// TwinCAT 3 PLC project liftConv
// ProgramVersion: 3.1.0.9
// libraries:
//   VisuElem3DPath, 3.5.6.0 (System)
//   VisuElemMeter, 3.5.6.0 (System)
//   VisuElems, 3.5.6.10 (System)
//   VisuElemsDateTime, 3.5.6.0 (System)
//   VisuElemsSpecialControls, 3.5.6.0 (System)
//   VisuElemsWinControls, 3.5.6.0 (System)
//   VisuElemTextEditor, 3.5.6.0 (System)
//   visuinputs, 3.5.6.0 (system)
//   VisuNativeControl, 3.5.6.0 (System)
//   Tc2_Standard, * (Beckhoff Automation GmbH)
//   Tc2_System, * (Beckhoff Automation GmbH)
//   Tc3_Interfaces, * (Beckhoff Automation GmbH)
//   Tc3_Module, * (Beckhoff Automation GmbH)
//   VisuDialogs, * (System)
// project tree:
//   / GlobalTextList.TcGTLO, PlcTask.TcTTO, Visualization Manager.TcVMO (not stored), VISU_TASK.TcTTO
//   GVLs/ GVL.TcGVL
//   POUs/ MAIN.TcPOU, outputFBD.TcPOU, NotUsed.TcPOU, Queues.TcPOU, resetOutputs.TcPOU, reset.TcPOU
//   VISUs/ TouchScreen.TcVIS
// real-time tasks:
//   TASK PlcTask: cycle T#10ms, priority 20, ADS port 350
//   TASK VISU_TASK: cycle T#100000us, priority 30, ADS port 351
// I/O:
//   DEVICE Device 1 (EtherCAT), AmsNetId 5.29.55.232.2.1
//     Term 1 (EK1100) [EK1100 EtherCAT Coupler (2A E-Bus)]
//       Term 2 (EL1008) [EL1008 8Ch. Dig. Input 24V, 3ms]
//       Term 3 (EL2008) [EL2008 8Ch. Dig. Output 24V, 0.5A]
//       Term 4 (EL3002) [EL3002 2Ch. Ana. Input +/-10V]
//       Term 5 (EL4002) [EL4002 2Ch. Ana. Output 0-10V, 12bit]
//       Term 6 (EL3124) [EL3124 4Ch. Ana. Input 4-20mA Diff.]
//       Term 7 (EL4024) [EL4024 4Ch. Ana. Output 4-20mA, 12bit]
//       Term 10 (EL9011) [EL9011 End Terminal]
//     Term 8 (EK1100) [EK1100 EtherCAT Coupler (2A E-Bus)]
//       Box 9 (BK1250)
// variable links:
//   liftConv/liftConv Instance <-> Device 1 (EtherCAT)/Term 1 (EK1100)/Term 2 (EL1008)
//     PlcTask Inputs/GVL.b{1..5} <-> Channel {1..5}/Input  (5 links)
//   liftConv/liftConv Instance <-> Device 1 (EtherCAT)/Term 8 (EK1100)/Box 9 (BK1250)
//     PlcTask Inputs/GVL.I_bInput11 <-> Term 4 (KL1104)/Channel 3/Input
//     PlcTask Inputs/GVL.I_bInput12 <-> Term 4 (KL1104)/Channel 4/Input
//     PlcTask Inputs/GVL.bottomLeft_IB <-> Term 4 (KL1104)/Channel 1/Input
//     PlcTask Inputs/GVL.bottomRight_IB <-> Term 3 (KL1104)/Channel 3/Input
//     PlcTask Inputs/GVL.leftLiftDownPosition_IB <-> Term 3 (KL1104)/Channel 2/Input
//     PlcTask Inputs/GVL.leftLiftOptical_IB <-> Term 2 (KL1104)/Channel 1/Input
//     PlcTask Inputs/GVL.leftLiftUpPosition_IB <-> Term 3 (KL1104)/Channel 1/Input
//     PlcTask Inputs/GVL.rightLiftDownPosition_IB <-> Term 2 (KL1104)/Channel 4/Input
//     PlcTask Inputs/GVL.rightLiftOptical_IB <-> Term 2 (KL1104)/Channel 2/Input
//     PlcTask Inputs/GVL.rightLiftUpPosition_IB <-> Term 2 (KL1104)/Channel 3/Input
//     PlcTask Inputs/GVL.topLeft_IB <-> Term 4 (KL1104)/Channel 2/Input
//     PlcTask Inputs/GVL.topRight_IB <-> Term 3 (KL1104)/Channel 4/Input
//     PlcTask Outputs/GVL.bottomBeltRight_OB <-> Term 7 (KL2114)/Channel 2/Output
//     PlcTask Outputs/GVL.leftLiftBeltLeft_OB <-> Term 6 (KL2114)/Channel 4/Output
//     PlcTask Outputs/GVL.leftLiftBeltRight_OB <-> Term 6 (KL2114)/Channel 3/Output
//     PlcTask Outputs/GVL.leftLiftDown_OB <-> Term 5 (KL2114)/Channel 2/Output
//     PlcTask Outputs/GVL.leftLiftUp_OB <-> Term 5 (KL2114)/Channel 1/Output
//     PlcTask Outputs/GVL.rightLiftBeltLeft_OB <-> Term 6 (KL2114)/Channel 1/Output
//     PlcTask Outputs/GVL.rightLiftBeltRight_OB <-> Term 6 (KL2114)/Channel 2/Output
//     PlcTask Outputs/GVL.rightLiftDown_OB <-> Term 5 (KL2114)/Channel 3/Output
//     PlcTask Outputs/GVL.rightLiftUp_OB <-> Term 5 (KL2114)/Channel 4/Output
//     PlcTask Outputs/GVL.topBeltLeft_OB <-> Term 7 (KL2114)/Channel 1/Output

CONFIGURATION liftConv
    RESOURCE PLC ON TwinCAT3
        TASK PlcTask(INTERVAL := T#10ms, PRIORITY := 20);
        TASK VISU_TASK(INTERVAL := T#100000us, PRIORITY := 30);
        PROGRAM MAIN WITH PlcTask : MAIN;
        PROGRAM VisuElems_Visu_Prg WITH VISU_TASK : VisuElems.Visu_Prg;
    END_RESOURCE
END_CONFIGURATION

// ---- GVLs/GVL.TcGVL
VAR_GLOBAL
//----------------------------------------------------------
//Inputs
	leftLiftOptical_IB AT %I*: BOOL; // DI 1 - Piece in the left lift
	rightLiftOptical_IB AT %I*: BOOL; // DI 2 - Piese in the right lift
	
//	I_bPieceLeftLift 		AT %I*: BOOL;	
//	I_bPieceRightLift 		AT %I*: BOOL;
	
	rightLiftDownPosition_IB AT %I*: BOOL;	// DI 3 - Right lift is bottom
	rightLiftUpPosition_IB AT %I*: BOOL;	// DI 4 - Right lift is up
	
//	I_bRightLiftBottom		AT %I*: BOOL;	
//	I_bRightLiftUp 			AT %I*: BOOL;
	
	leftLiftDownPosition_IB AT %I*: BOOL;	// DI 5 - Left lift is down
	leftLiftUpPosition_IB AT %I*: BOOL;	// DI 6 - Left lift is up	
	
//	I_bLeftLiftDown		AT %I*: BOOL;	
//	I_bLeftLiftUp			AT %I*: BOOL;	
	
	bottomRight_IB AT %I*: BOOL;		// DI 7 - Piece on low belt right side
	topRight_IB AT %I*: BOOL;			// DI 8 - Piece on top belt right side
	
//	I_bLowBeltRight			AT %I*: BOOL;	
//	I_bTopBeltRight			AT %I*: BOOL;
	
	bottomLeft_IB AT %I*: BOOL;		// DI 9 - Piece on low belt left side
	topLeft_IB AT %I*: BOOL;		// DI 10 - Piece on top belt left side
	
//	I_bLowBeltLeft			AT %I*: BOOL;	
//	I_bTopBeltLeft			AT %I*: BOOL;	
	
	I_bInput11 				AT %I*: BOOL;	// DI 11 - Empty
	I_bInput12 				AT %I*: BOOL;   // DI 12 - Empty

	b1 AT %I*: BOOL;
	b2 AT %I*: BOOL;
	b3 AT %I*: BOOL;
	b4 AT %I*: BOOL;
	b5 AT %I*: BOOL;
//----------------------------------------------------------
//Outputs
	
	leftLiftUp_OB	AT %Q*: BOOL; 	// DO 1 - Left Lift up
	leftLiftDown_OB	AT %Q*: BOOL;	// DO 2 - Left Lift down
	
//	O_bLeftLiftUp 			AT %Q*: BOOL;
//	O_bLeftLiftDown 		AT %Q*: BOOL;

	rightLiftDown_OB		AT %Q*: BOOL;	 // DO 3 - Right Lift down
	rightLiftUp_OB AT %Q*: BOOL;			// DO 4 - Right Lift up
	
//	O_bRightLiftDown		AT %Q*: BOOL;	
//	O_bRightLiftUp			AT %Q*: BOOL;	
	
	rightLiftBeltLeft_OB 	AT %Q*: BOOL; 	// DO 5 - Lift Right belt left
	rightLiftBeltRight_OB 	AT %Q*: BOOL;	// DO 6 - Lift Right belt right
	
//	O_bRightLiftBeltLeft	AT %Q*: BOOL;	
//	O_bRightLiftBeltRight	AT %Q*: BOOL;

	leftLiftBeltRight_OB 	AT %Q*: BOOL;	// DO 7 - Lift Left belt right
	leftLiftBeltLeft_OB 	AT %Q*: BOOL;	// DO 8 - Lift Left belt left
	
//	O_bLeftLiftBeltRight	AT %Q*: BOOL;	
//	O_bLeftLiftBeltLeft		AT %Q*: BOOL;	
	
	topBeltLeft_OB 	AT %Q*: BOOL;	// DO 9 - Top belt left
	bottomBeltRight_OB 	AT %Q*: BOOL;	// DO 10 - Low belt right
	
//	O_bTopBeltLeft 			AT %Q*: BOOL;	
//	O_bLowBeltRight 			AT %Q*: BOOL;

	topBeltRight_OB AT %Q*: BOOL;	// DO 11 - Top belt right
	lowBeltLeft_OB AT %Q*: BOOL;	// DO 12 - Low belt left
 	
//	O_bTopBeltRight			AT %Q*: BOOL;	
//	O_bLowBeltLeft			AT %Q*: BOOL; 




//----------------------------------------------------------
//Memory

	running : BOOL;
	resetAll : BOOL;
	trowingObjectOut : BOOL;
	
	
	obj1 : INT;
	obj2 : INT;
	obj3 : INT;
	obj4 : INT;	
	obj : ARRAY[1..5] OF INT;

	
	topRightLiftExp : INT;
	topRightLiftExpArr : ARRAY[1..5] OF INT;
	topRightExp : INT;
	topRightExpArr : ARRAY[1..5] OF INT;
	topLeftExp : INT;
	topLeftExpArr : ARRAY[1..5] OF INT;
	topLeftLiftExp : INT;
	topLeftLiftExpArr : ARRAY[1..5] OF INT;
	bottomLeftLiftExp : INT;
	bottomLeftLiftExpArr : ARRAY[1..5] OF INT;
	bottomLeftExp : INT;
	bottomLeftExpArr : ARRAY[1..5] OF INT;
	bottomRightExp : INT;
	bottomRightExpArr : ARRAY[1..5] OF INT;
	bottomRightLiftExp : INT;
	bottomRightLiftExpArr : ARRAY[1..5] OF INT;
	
	ERR: INT;
	resetError: BOOL;
	auto: BOOL;
	textMA : WSTRING;
	errMessage : WSTRING;
END_VAR

// ---- POUs/MAIN.TcPOU
PROGRAM MAIN
VAR
	queues : Queues;
	auto_lastCycle: BOOL;
	myvar: INT;
	initiated: BOOL;
	ERR_lastCycle: INT;
END_VAR

VAR_INPUT
END_VAR

IF ERR = 0 THEN
	queues();
	IF auto THEN
		outputFBD();	
	END_IF
ELSE
	//error handling
	resetOutputs();
	
	IF ERR <> ERR_lastCycle THEN
		CASE ERR OF
			1:
				errMessage := "1: Unexpected object on the right of top belt";
			2:
				errMessage := "2: Unexpected object on the left of top belt";
			3:
				errMessage := "3: Unexpected object on the left lift (top position)";
			4:
				errMessage := "3: Unexpected object on the left lift (bottom position)";
			5:
				errMessage := "5: Unexpected object on the left of bottom belt";
			6:
				errMessage := "6: Unexpected object on the right of bottom belt";
			7:
				errMessage := "7: Unexpected object on the right lift (bottom position)";
			8:
				errMessage := "8: Cannot accept new object. Over capacity.";

		ELSE
			errMessage := INT_TO_WSTRING(ERR);	
		END_CASE
			
	END_IF
	ERR_lastCycle := ERR;
END_IF


IF resetAll OR b5 THEN
	reset();
END_IF

IF resetError OR b5 THEN
	ERR :=0;
	auto := False;
	resetError := FALSE;
END_IF


IF auto <> auto_lastCycle THEN
	IF auto THEN
		textMA := "AUTOMATIC";
	ELSE
		textMA :="MANUAL";		
	END_IF	
END_IF
IF NOT auto AND auto_lastCycle THEN
	resetOutputs();
END_IF
auto_lastCycle := auto;

IF NOT initiated THEN
	textMA := "MANUAL";
END_IF
initiated := TRUE;

END_PROGRAM

// ---- POUs/Queues.TcPOU
FUNCTION_BLOCK Queues
VAR_INPUT
END_VAR
VAR_OUTPUT
END_VAR
VAR
	fcT1: TOF;
	fcT2: TOF;
	fcT3: TOF;
	fcT4: TOF;
	fcT5: TOF;
	fcT6: TOF;
	fcT7: TOF;
	fcT8: TOF;
	onDelayT9 : TON;
	onDelayT10 : TON;
	
	T1: BOOL;
	T2: BOOL;
	T3: BOOL;
	T4: BOOL;
	T5: BOOL;
	T6: BOOL;
	T7: BOOL;
	T8: BOOL;
	T9: BOOL;
	T10: BOOL;

	goAroundCycles : INT := 2;
	trowObjectOut: BOOL;

	T9c2: BOOL;
	T10c2: BOOL;

	assigned: BOOL; //these are used in first paragraph
	i: INT;

END_VAR

//----------------------------------------------------------	
//object entrance location top righ on lift.

IF rightLiftOptical_IB AND rightLiftUpPosition_IB AND NOT T1 THEN
	IF topRightLiftExp = 0 THEN
		assigned := FALSE;
		i := 1;
		WHILE i<5 AND NOT assigned DO
			IF obj[i] = 0 THEN
				obj[i] := 1;
				assigned := TRUE;
			ELSE
				i := i + 1;
			END_IF
		END_WHILE
		IF NOT assigned THEN
			ERR:=8;
			RETURN;
		END_IF
		topRightExp := topRightExp+1;
		topRightExpArr[topRightExp]:= i;
	ELSE
			topRightExp := topRightExp+1;
			topRightExpArr[topRightExp]:= topRightLiftExpArr[1];
			topRightLiftExp := 0;
			topRightLiftExpArr[1] := 0;					
	END_IF

END_IF
fcT1(IN:=(rightLiftOptical_IB AND rightLiftUpPosition_IB), PT:=T#1S, Q=>T1);

//----------------------------------------------------------
//object on top right conveyor sensor

IF topRight_IB  AND NOT T2 THEN
	IF topRightExp = 0 THEN
		ERR := 1;
		return;
	ELSE
		topRightExp := topRightExp -1;	
		topLeftExp := topLeftExp +1;
		topLeftExpArr[topLeftExp] := topRightExpArr[1];
		topRightExpArr[1] := topRightExpArr[2];
		topRightExpArr[2] := topRightExpArr[3];
		topRightExpArr[3] := topRightExpArr[4];
		topRightExpArr[4] := topRightExpArr[5];
		topRightExpArr[5] := 0;		
	END_IF
END_IF
fcT2(IN:=topRight_IB , PT:=T#300MS, Q=>T2);

//----------------------------------------------------------
//object on top left conveyor sensor

IF topLeft_IB AND NOT T3 THEN
	IF topLeftExp = 0 THEN
		ERR := 2;
		RETURN;
	ELSE
		topLeftExp := topLeftExp -1;	
		topLeftLiftExp := topLeftLiftExp +1;
		topLeftLiftExpArr[topLeftLiftExp] :=topLeftExpArr[1];
		topLeftExpArr[1] := topLeftExpArr[2];
		topLeftExpArr[2] := topLeftExpArr[3];
		topLeftExpArr[3] := topLeftExpArr[4];
		topLeftExpArr[4] := topLeftExpArr[5];
		topLeftExpArr[5] := 0;		
	END_IF
END_IF
fcT3(IN:=topLeft_IB , PT:=T#300MS, Q=>T3);

//----------------------------------------------------------
//object detected on left lift when the lift is up

fcT4(IN:=(leftLiftUpPosition_IB AND leftLiftOptical_Ib), PT:=T#100MS, Q=>T4);
onDelayT9( IN:= T4,  PT:= T#1500MS, Q => T9);
IF T9 AND NOT T9c2 THEN
	IF topLeftLiftExp = 0 THEN
		ERR := 3;
		RETURN;
	ELSE
		topLeftLiftExp := topLeftLiftExp - 1;
		bottomLeftLiftExp := bottomLeftLiftExp +1;
		bottomLeftLiftExpArr[bottomLeftLiftExp] := topLeftLiftExpArr[1];
		topLeftLiftExpArr[1] := topLeftLiftExpArr[2];
		topLeftLiftExpArr[2] := topLeftLiftExpArr[3];
		topLeftLiftExpArr[3] := topLeftLiftExpArr[4];
		topLeftLiftExpArr[4] := topLeftLiftExpArr[5];
		topLeftLiftExpArr[5] := 0;
	END_IF
END_IF
T9c2 := T9;

//----------------------------------------------------------
//object detected on left lift when the lift is down

IF leftLiftDownPosition_IB AND leftLiftOptical_IB AND NOT T5 THEN
	IF bottomLeftLiftExp = 0 THEN
		ERR := 4;
	ELSE
		bottomLeftLiftExp := 0;
		bottomLeftExp := bottomLeftExp +1;
		bottomLeftExpArr[bottomLeftExp] := bottomLeftLiftExpArr[1];
		bottomLeftLiftExpArr[1] := 0;
	END_IF
END_IF
fcT5(IN:=(leftLiftDownPosition_IB AND leftLiftOptical_IB), PT:=T#300MS, Q=>T5);


//----------------------------------------------------------
//object detected on bottom belt left sensor

IF bottomLeft_IB AND NOT T5 THEN
	IF bottomLeftExp = 0 THEN
		ERR := 5;
		RETURN;
	ELSE
		bottomLeftExp := bottomLeftExp - 1;
		bottomRightExp := bottomRightExp +1;
		bottomRightExpArr[bottomRightExp] := bottomLeftExpArr[1];
		bottomLeftExpArr[1] := bottomLeftExpArr[2];
		bottomLeftExpArr[2] := bottomLeftExpArr[3];
		bottomLeftExpArr[3] := bottomLeftExpArr[4];
		bottomLeftExpArr[4] := bottomLeftExpArr[5];
		bottomLeftExpArr[5] := 0;
	END_IF
END_IF
fcT5(IN:= bottomLeft_IB, PT:=T#300MS, Q=>T5);

//----------------------------------------------------------
//object detected on bottom belt right sensor

IF bottomRight_IB AND NOT T6 THEN
	IF bottomRightExp = 0 THEN
		ERR := 6;
		RETURN;
	ELSE
		bottomRightExp := bottomRightExp - 1;
		bottomRightLiftExp := bottomRightLiftExp +1;
		bottomRightLiftExpArr[bottomRightLiftExp] := bottomRightExpArr[1];
		bottomRightExpArr[1] := bottomRightExpArr[2];
		bottomRightExpArr[2] := bottomRightExpArr[3];
		bottomRightExpArr[3] := bottomRightExpArr[4];
		bottomRightExpArr[4] := bottomRightExpArr[5];
		bottomRightExpArr[5] := 0;
	END_IF
END_IF
fcT6(IN:= bottomRight_IB, PT:=T#300MS, Q=>T6);

//----------------------------------------------------------
//object detected on right lift sensor when the lift is down


fcT7(IN:=(rightLiftDownPosition_IB AND rightLiftOptical_IB), PT:=T#100MS, Q=>T7);
onDelayT10(IN:= T7, PT:=T#1500MS, Q=>T10);
IF (T10 AND NOT T10c2) AND NOT trowingObjectOut THEN
	IF bottomRightLiftExp = 0 THEN
		ERR := 7;
		RETURN;
	ELSE
		bottomRightLiftExp := bottomRightLiftExp - 1;
		IF obj[bottomRightLiftExpArr[1]] >= goAroundCycles THEN
			obj[bottomRightLiftExpArr[1]] :=0;
			trowObjectOut := TRUE;
		ELSE
			obj[bottomRightLiftExpArr[1]] :=1+obj[bottomRightLiftExpArr[1]];
			topRightLiftExp := topRightLiftExp +1;
			topRightLiftExpArr[topRightLiftExp] := bottomRightLiftExpArr[1];
		END_IF
		bottomRightLiftExpArr[1] := bottomRightLiftExpArr[2];
		bottomRightLiftExpArr[2] := bottomRightLiftExpArr[3];
		bottomRightLiftExpArr[3] := bottomRightLiftExpArr[4];
		bottomRightLiftExpArr[4] := bottomRightLiftExpArr[5];
		bottomRightLiftExpArr[5] := 0;
	END_IF		

END_IF
T10c2 := T10;
fcT8(IN:=(trowObjectOut or (trowingObjectOut and rightLiftOptical_IB)), PT:=T#2S, Q=>TrowingObjectOut);
trowObjectOut := FALSE;

END_FUNCTION_BLOCK

// ---- POUs/outputFBD.TcPOU
FUNCTION outputFBD : INT
VAR_INPUT
END_VAR
VAR
	bottomBeltLeft_OB: BOOL;
END_VAR
VAR // added by the converter: edge detectors and wires of the graphical bodies
    _w1, _w2 : BOOL;
END_VAR

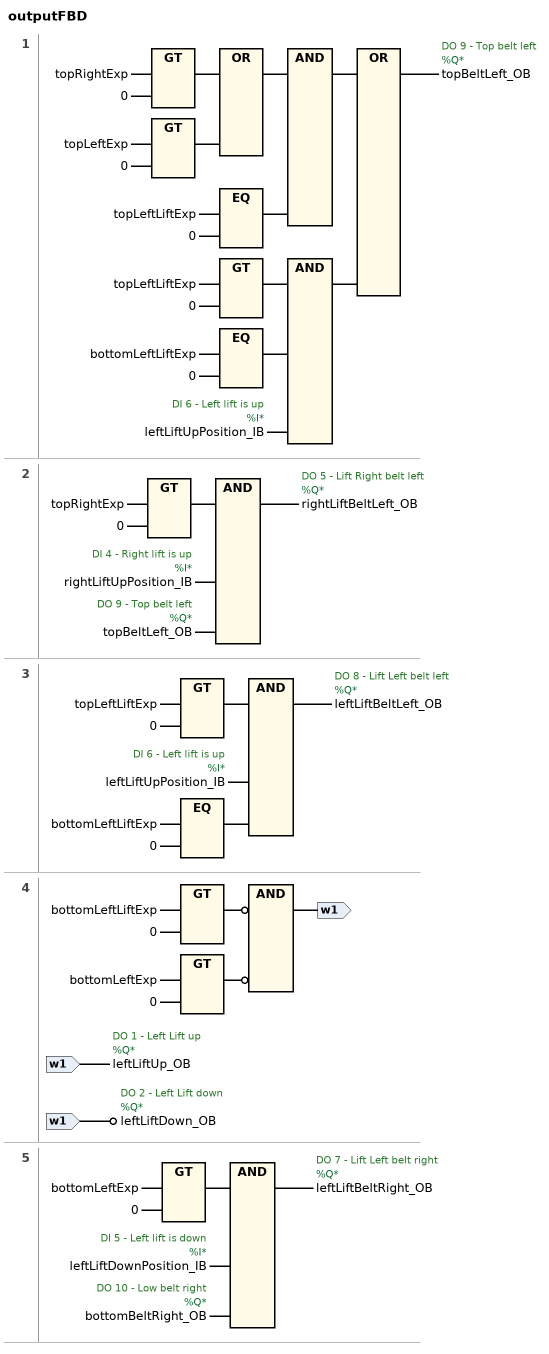
// NETWORK 1
//   leftLiftUpPosition_IB: DI 6 - Left lift is up | AT %I*
//   topBeltLeft_OB: DO 9 - Top belt left | AT %Q*
topBeltLeft_OB := (topRightExp > 0 OR topLeftExp > 0) AND topLeftLiftExp = 0 OR topLeftLiftExp > 0 AND bottomLeftLiftExp = 0 AND leftLiftUpPosition_IB;

// NETWORK 2
//   rightLiftUpPosition_IB: DI 4 - Right lift is up | AT %I*
//   topBeltLeft_OB: DO 9 - Top belt left | AT %Q*
//   rightLiftBeltLeft_OB: DO 5 - Lift Right belt left | AT %Q*
rightLiftBeltLeft_OB := topRightExp > 0 AND rightLiftUpPosition_IB AND topBeltLeft_OB;

// NETWORK 3
//   leftLiftUpPosition_IB: DI 6 - Left lift is up | AT %I*
//   leftLiftBeltLeft_OB: DO 8 - Lift Left belt left | AT %Q*
leftLiftBeltLeft_OB := topLeftLiftExp > 0 AND leftLiftUpPosition_IB AND bottomLeftLiftExp = 0;

// NETWORK 4
//   leftLiftUp_OB: DO 1 - Left Lift up | AT %Q*
//   leftLiftDown_OB: DO 2 - Left Lift down | AT %Q*
_w1 := NOT (bottomLeftLiftExp > 0) AND NOT (bottomLeftExp > 0);
leftLiftUp_OB := _w1;
leftLiftDown_OB := NOT _w1;

// NETWORK 5
//   leftLiftDownPosition_IB: DI 5 - Left lift is down | AT %I*
//   bottomBeltRight_OB: DO 10 - Low belt right | AT %Q*
//   leftLiftBeltRight_OB: DO 7 - Lift Left belt right | AT %Q*
leftLiftBeltRight_OB := bottomLeftExp > 0 AND leftLiftDownPosition_IB AND bottomBeltRight_OB;

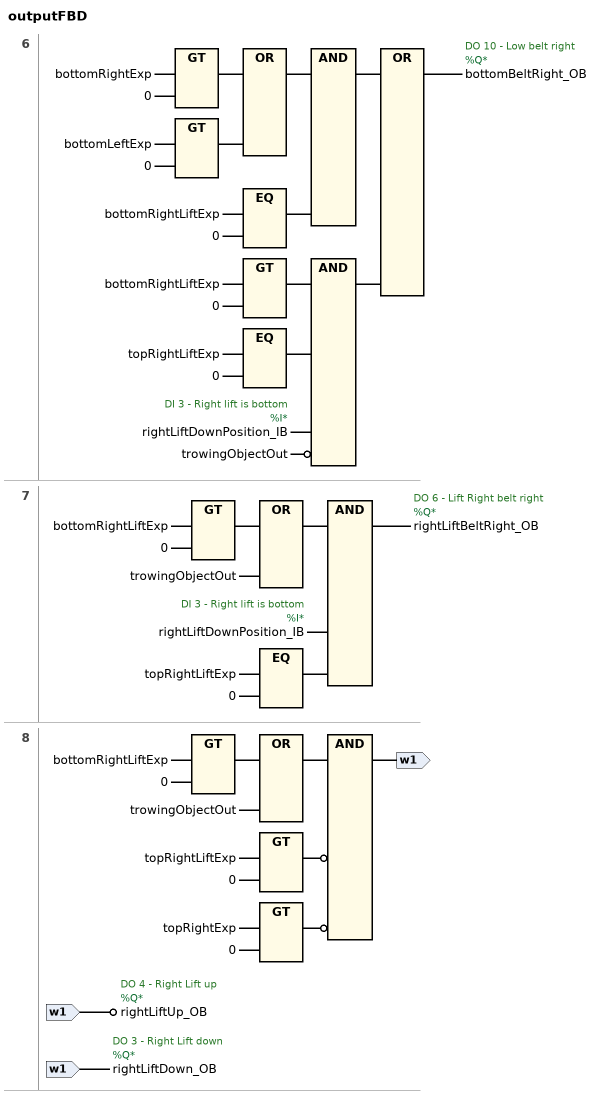
// NETWORK 6
//   rightLiftDownPosition_IB: DI 3 - Right lift is bottom | AT %I*
//   bottomBeltRight_OB: DO 10 - Low belt right | AT %Q*
bottomBeltRight_OB := (bottomRightExp > 0 OR bottomLeftExp > 0) AND bottomRightLiftExp = 0 OR bottomRightLiftExp > 0 AND topRightLiftExp = 0 AND rightLiftDownPosition_IB AND NOT trowingObjectOut;

// NETWORK 7
//   rightLiftDownPosition_IB: DI 3 - Right lift is bottom | AT %I*
//   rightLiftBeltRight_OB: DO 6 - Lift Right belt right | AT %Q*
rightLiftBeltRight_OB := (bottomRightLiftExp > 0 OR trowingObjectOut) AND rightLiftDownPosition_IB AND topRightLiftExp = 0;

// NETWORK 8
//   rightLiftUp_OB: DO 4 - Right Lift up | AT %Q*
//   rightLiftDown_OB: DO 3 - Right Lift down | AT %Q*
_w2 := (bottomRightLiftExp > 0 OR trowingObjectOut) AND NOT (topRightLiftExp > 0) AND NOT (topRightExp > 0);
rightLiftUp_OB := NOT _w2;
rightLiftDown_OB := _w2;

END_FUNCTION

// ---- POUs/resetOutputs.TcPOU
FUNCTION resetOutputs : int
VAR_INPUT
END_VAR
VAR
END_VAR

trowingObjectOut := 0;
leftLiftUp_OB := 0;
leftLiftDown_OB := 0;
rightLiftDown_OB := 0;
rightLiftUp_OB := 0;
rightLiftBeltLeft_OB := 0;
rightLiftBeltRight_OB := 0;
leftLiftBeltRight_OB := 0;
leftLiftBeltLeft_OB  := 0;
topBeltLeft_OB  := 0;
bottomBeltRight_OB := 0;
topBeltRight_OB := 0;
lowBeltLeft_OB := 0;

END_FUNCTION

// ---- POUs/reset.TcPOU
FUNCTION reset : int
VAR_INPUT
END_VAR
VAR
	i: INT;
END_VAR

FOR i:=1 TO 5 BY 1 DO
	topRightLiftExpArr[i] := 0;
	topRightExpArr[i] := 0;
	topLeftExpArr[i] := 0;
	topLeftLiftExpArr[i] := 0;
	bottomLeftLiftExpArr[i] := 0;
	bottomLeftExpArr[i] := 0;
	bottomRightExpArr[i] := 0;
	bottomRightLiftExpArr[i] := 0;
	obj[i] := 0;
END_FOR

topRightLiftExp := 0;
topRightExp := 0;
topLeftExp := 0;
topLeftLiftExp := 0;
bottomLeftLiftExp := 0;
bottomLeftExp := 0;
bottomRightExp := 0;
bottomRightLiftExp := 0;


trowingObjectOut := 0;
leftLiftUp_OB := 0;
leftLiftDown_OB := 0;
rightLiftDown_OB := 0;
rightLiftUp_OB := 0;
rightLiftBeltLeft_OB := 0;
rightLiftBeltRight_OB := 0;
leftLiftBeltRight_OB := 0;
leftLiftBeltLeft_OB  := 0;
topBeltLeft_OB  := 0;
bottomBeltRight_OB := 0;
topBeltRight_OB := 0;
lowBeltLeft_OB := 0;
ERR := 0;
resetAll := FALSE;

END_FUNCTION

// ---- POUs/NotUsed.TcPOU
FUNCTION NotUsed : int
VAR_INPUT
END_VAR
VAR
END_VAR


//----------------------------------------------------------
//Output control depending on queues and lift positions

IF (topRightExp>0 OR topLeftExp>0) AND topLeftLiftExp = 0 THEN
	topBeltLeft_OB :=TRUE;
END_IF

IF topRightExp>0 AND rightLiftUpPosition_IB AND topBeltLeft_OB THEN
	rightLiftBeltLeft_OB := TRUE;
ELSE
	rightLiftBeltLeft_OB := FALSE;
END_IF

IF topLeftLiftExp > 0 AND bottomLeftLiftExp = 0 AND leftLiftUpPosition_IB  THEN
	leftLiftBeltLeft_OB := TRUE;
ELSE
	leftLiftBeltLeft_OB := FALSE;
END_IF

IF bottomLeftLiftExp >1  THEN
	leftLiftDown_OB := TRUE;
	leftLiftUp_OB := FALSE;
END_IF

IF bottomLeftExp > 1 AND bottomRightLiftExp=0 THEN
	leftLiftBeltLeft_OB := TRUE;
	bottomBeltRight_OB :=TRUE;
END_IF

IF bottomLeftExp = 0  AND bottomLeftLiftExp = 0 THEN
	leftLiftBeltLeft_OB := FALSE;
	leftLiftUp_OB := TRUE;
	leftLiftDown_OB := FALSE;
END_IF

IF bottomRightExp > 0 AND (bottomRightLiftExp=0 AND NOT trowingObjectOut) THEN
	bottomBeltRight_OB := TRUE;
END_IF

IF bottomRightLiftExp > 0 AND topRightExp = 0 AND topRightLiftExp = 0 AND rightLiftUpPosition_IB THEN
	rightLiftDown_OB := TRUE;
	rightLiftUp_OB := FALSE;
END_IF

IF bottomRightLiftExp > 0 AND topRightExp = 0 AND rightLiftDownPosition_IB THEN
	rightLiftBeltRight_OB := TRUE;
	bottomBeltRight_OB := TRUE;
END_IF

IF topRightLiftExp = 0 AND NOT trowingObjectOut THEN
	rightLiftBeltRight_OB := FALSE;
	rightLiftUp_OB :=TRUE;
	rightLiftDown_OB :=FALSE;
END_IF

IF topRightLiftExp = 1 THEN
	rightLiftBeltRight_OB := FALSE;
	bottomBeltRight_OB :=FALSE;
	rightLiftUp_OB :=TRUE;
	rightLiftDown_OB :=FALSE;
END_IF

IF trowingObjectOut THEN
	rightLiftBeltRight_OB := TRUE;
	bottomBeltRight_OB := FALSE;
END_IF

IF bottomRightLiftExp > 1 AND NOT rightLiftDownPosition_IB THEN
	bottomBeltRight_OB := FALSE;
END_IF

IF resetAll THEN
	reset();
END_IF

END_FUNCTION

// ---- GlobalTextList.TcGTLO
TEXTLIST GlobalTextList
  49 = ' %s'
  55 = ' bottomLeft %d'
  57 = ' bottomRightLift %d'
  16 = '%d'
  41 = '%s'
  38 = '++++++++++++++++++++++++++++++++++++++++++++++++++++++++++++++++++++++++++++++++++++++++++++++++++++++'
  54 = 'bottomLeftLift %d'
  56 = 'bottomRight %d'
  40 = 'Clear'
  58 = 'Cycle : % d'
  31 = 'ERR. %d'
  32 = 'exp on bottomLeft %d'
  22 = 'exp on bottomLeft%d'
  21 = 'exp on bottomLeftLift %d'
  33 = 'exp on bottomRight %d'
  23 = 'exp on bottomRight%d'
  35 = 'exp on bottomRightLift %d'
  24 = 'exp on bottomRightLift%d'
  34 = 'exp on bottomRightLiftd'
  37 = 'exp on topLeft %d'
  19 = 'exp on topLeft%d'
  36 = 'exp on topLeftLift  %d'
  20 = 'exp on topLeftLift %d'
  18 = 'exp on topRighLift %d'
  8 = 'expecting     %d    :  %d d d d d on topRight'
  9 = 'expecting     %d    :  d d d d d on topRight'
  7 = 'expecting     %d    : d d d d d on topRight'
  4 = 'expecting     %d : %d %d %d %d %d on topRight'
  5 = 'expecting     %d : %d d d d d on topRight'
  6 = 'expecting     %d : d d d d d on topRight'
  10 = 'expecting     %i    :  d d d d d on topRight'
  2 = 'expecting     %i : %i %i %i %i %i'
  3 = 'expecting     %i : %i %i %i %i %i on topRight'
  13 = 'expecting %d'
  12 = 'expecting %d    :  %d d d d d on topRight'
  11 = 'expecting %d    :  d d d d d on topRight'
  14 = 'expecting %d %d'
  15 = 'expecting on topRigh %d'
  17 = 'expecting on topRighLift %d'
  25 = 'obj1 cycles: %d'
  44 = 'obj1 on cycle %d'
  26 = 'obj2 cycles: %d'
  45 = 'obj2 on cycle %d'
  27 = 'obj3 cycles: %d'
  46 = 'obj3 on cycle %d'
  47 = 'obj4 cycle %d'
  28 = 'obj4 cycles: %d'
  48 = 'obj4 on cycle %d'
  59 = 'Object n.1'
  43 = 'Objects:'
  30 = 'Reset'
  60 = 'Reset all'
  39 = 'Reset Error'
  42 = 'textMA[auto]'
  52 = 'topLeft %d'
  53 = 'topLeftLift  %d'
  51 = 'topRigh %d'
  50 = 'topRighLift %d'
  29 = 'trowing out'
  1 = '\\n%i\\n%i\\n%i\\n%i\\n%i\\nexp %i'
  0 = '\\nexp %i'
END_TEXTLIST

// ---- VISUs/TouchScreen.TcVIS
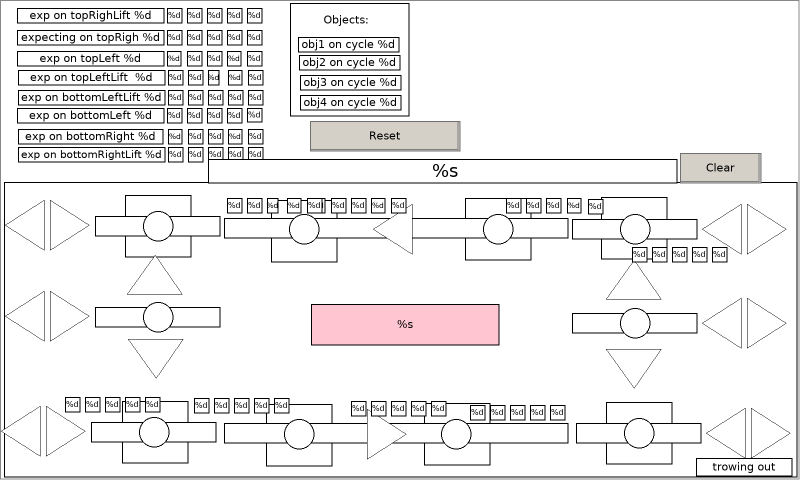
VISUALIZATION TouchScreen  // 800x480
    Rectangle (4,182 793x295), colour toggle: ERR <> 0, invisible if: ERR = 0
    Rectangle (601,197 66x62), colour toggle: ERR <> 0, invisible if: ERR <> 8
    Rectangle (606,402 66x62), colour toggle: ERR <> 0, invisible if: ERR <> 7
    Rectangle (424,403 66x62), colour toggle: ERR <> 0, invisible if: ERR <> 6
    Rectangle (266,404 66x62), colour toggle: ERR <> 0, invisible if: ERR <> 5
    Rectangle (122,401 66x62), colour toggle: ERR <> 0, invisible if: ERR <> 4
    Rectangle (125,195 66x62), colour toggle: ERR <> 0, invisible if: ERR <> 3
    Rectangle (271,200 66x62), colour toggle: ERR <> 0, invisible if: ERR <> 2
    RoundedRectangle (224,423 344x20)
    Rectangle (465,198 66x62), colour toggle: ERR <> 0, invisible if: ERR <> 1
    RoundedRectangle (224,218 344x20)
    RoundedRectangle (572,219 125x20), invisible if: rightLiftUpPosition_IB <> True
    Rectangle (290,3 119x113)
    Rectangle (17,30 147x15), "expecting on topRigh %d", text variable: GVL.topRightExp
    Rectangle (167,30 15x15), "%d", text variable: GVL.topRightExpArr[1], invisible if: GVL.topRightExpArr[1]=0
    Rectangle (187,30 15x15), "%d", text variable: GVL.topRightExpArr[2], invisible if: GVL.topRightExpArr[2]=0
    Rectangle (207,30 15x15), "%d", text variable: GVL.topRightExpArr[3], invisible if: GVL.topRightExpArr[3]=0
    Rectangle (227,30 15x15), "%d", text variable: GVL.topRightExpArr[4], invisible if: GVL.topRightExpArr[4]=0
    Rectangle (247,30 15x15), "%d", text variable: GVL.topRightExpArr[5], invisible if: GVL.topRightExpArr[5]=0
    Rectangle (17,8 147x15), "exp on topRighLift %d", text variable: GVL.topRightLiftExp
    Rectangle (167,8 15x15), "%d", text variable: GVL.topRightLiftExpArr[1], invisible if: GVL.topRightLiftExpArr[1]=0
    Rectangle (187,8 15x15), "%d", text variable: GVL.topRightLiftExpArr[2], invisible if: GVL.topRightLiftExpArr[2]=0
    Rectangle (207,8 15x15), "%d", text variable: GVL.topRightLiftExpArr[3], invisible if: GVL.topRightLiftExpArr[3]=0
    Rectangle (227,8 15x15), "%d", text variable: GVL.topRightLiftExpArr[4], invisible if: GVL.topRightLiftExpArr[4]=0
    Rectangle (247,8 15x15), "%d", text variable: GVL.topRightLiftExpArr[5], invisible if: GVL.topRightLiftExpArr[5]=0
    Rectangle (17,51 147x15), "exp on topLeft %d", text variable: GVL.topLeftExp
    Rectangle (167,51 14x15), "%d", text variable: GVL.topLeftExpArr[1], invisible if: GVL.topLeftExpArr[1] = 0
    Rectangle (187,51 15x15), "%d", text variable: GVL.topLeftExpArr[2], invisible if: GVL.topLeftExpArr[2]=0
    Rectangle (207,51 15x15), "%d", text variable: GVL.topLeftExpArr[3], invisible if: GVL.topLeftExpArr[3]=0
    Rectangle (227,51 14x15), "%d", text variable: GVL.topLeftExpArr[4], invisible if: GVL.topLeftExpArr[4]=0
    Rectangle (247,51 15x15), "%d", text variable: GVL.topLeftExpArr[5], invisible if: GVL.topLeftExpArr[5]=0
    Rectangle (18,70 147x15), "exp on topLeftLift %d", text variable: GVL.topLeftLiftExp
    Rectangle (168,70 15x15), "%d", text variable: GVL.topLeftLiftExpArr[1], invisible if: GVL.topLeftLiftExpArr[1]=0
    Rectangle (188,70 15x15), "%d", text variable: GVL.topLeftLiftExpArr[2], invisible if: GVL.topLeftLiftExpArr[2]=0
    Rectangle (208,70 11x15), "%d", text variable: GVL.topLeftLiftExpArr[3], invisible if: GVL.topLeftLiftExpArr[3]=0
    Rectangle (228,70 14x15), "%d", text variable: GVL.topLeftLiftExpArr[4], invisible if: GVL.topLeftLiftExpArr[4]=0
    Rectangle (248,70 15x15), "%d", text variable: GVL.topLeftLiftExpArr[5], invisible if: GVL.topLeftLiftExpArr[5]=0
    Rectangle (18,90 147x15), "exp on bottomLeftLift %d", text variable: GVL.bottomLeftLiftExp
    Rectangle (168,90 15x15), "%d", text variable: GVL.bottomLeftLiftExpArr[1], invisible if: GVL.bottomLeftLiftExpArr[1]=0
    Rectangle (188,90 15x15), "%d", text variable: GVL.bottomLeftLiftExpArr[2], invisible if: GVL.bottomLeftLiftExpArr[2]=0
    Rectangle (208,90 15x15), "%d", text variable: GVL.bottomLeftLiftExpArr[3], invisible if: GVL.bottomLeftLiftExpArr[3]=0
    Rectangle (228,90 15x15), "%d", text variable: GVL.bottomLeftLiftExpArr[4], invisible if: GVL.bottomLeftLiftExpArr[4] = 0
    Rectangle (248,90 15x15), "%d", text variable: GVL.bottomLeftLiftExpArr[5], invisible if: GVL.bottomLeftLiftExpArr[5]=0
    Rectangle (17,108 147x15), "exp on bottomLeft %d", text variable: GVL.bottomLeftExp
    Rectangle (167,108 15x15), "%d", text variable: GVL.bottomLeftExpArr[1], invisible if: GVL.bottomLeftExpArr[1]=0
    Rectangle (187,108 15x15), "%d", text variable: GVL.bottomLeftExpArr[2], invisible if: GVL.bottomLeftExpArr[2]=0
    Rectangle (207,108 15x15), "%d", text variable: GVL.bottomLeftExpArr[3], invisible if: GVL.bottomLeftExpArr[3]=0
    Rectangle (227,108 15x15), "%d", text variable: GVL.bottomLeftExpArr[4], invisible if: GVL.bottomLeftExpArr[4]=0
    Rectangle (247,108 15x14), "%d", text variable: GVL.bottomLeftExpArr[5], invisible if: GVL.bottomLeftExpArr[5]=0
    Rectangle (18,129 145x15), "exp on bottomRight %d", text variable: GVL.bottomRightExp
    Rectangle (168,129 14x15), "%d", text variable: GVL.bottomRightExpArr[1], invisible if: GVL.bottomRightExpArr[1]=0
    Rectangle (188,129 15x15), "%d", text variable: GVL.bottomRightExpArr[2], invisible if: GVL.bottomRightExpArr[2]=0
    Rectangle (208,129 15x15), "%d", text variable: GVL.bottomRightExpArr[3], invisible if: GVL.bottomRightExpArr[3]=0
    Rectangle (228,129 14x15), "%d", text variable: GVL.bottomRightExpArr[4], invisible if: GVL.bottomRightExpArr[4]=0
    Rectangle (248,129 15x15), "%d", text variable: GVL.bottomRightExpArr[5], invisible if: GVL.bottomRightExpArr[5]=0
    Rectangle (18,147 147x15), "exp on bottomRightLift %d", text variable: GVL.bottomRightLiftExp
    Rectangle (168,147 15x15), "%d", text variable: GVL.bottomRightLiftExpArr[1], invisible if: GVL.bottomRightLiftExpArr[1]=0
    Rectangle (188,147 15x15), "%d", text variable: GVL.bottomRightLiftExpArr[2], invisible if: GVL.bottomRightLiftExpArr[2]=0
    Rectangle (208,147 15x15), "%d", text variable: GVL.bottomRightLiftExpArr[3], invisible if: GVL.bottomRightLiftExpArr[3] = 0
    Rectangle (228,147 15x15), "%d", text variable: GVL.bottomRightLiftExpArr[4], invisible if: GVL.bottomRightLiftExpArr[4] = 0
    Rectangle (248,147 15x15), "%d", text variable: GVL.bottomRightLiftExpArr[5], invisible if: GVL.bottomRightLiftExpArr[5] = 0
    Rectangle (299,55 101x15), "obj2 on cycle %d", text variable: GVL.obj[2], invisible if: GVL.obj[2] = 0
    Rectangle (298,37 101x15), "obj1 on cycle %d", text variable: GVL.obj[1], invisible if: GVL.obj[1]=0
    Rectangle (300,75 101x15), "obj3 on cycle %d", text variable: GVL.obj[3], invisible if: GVL.obj[3] = 0
    Rectangle (300,95 101x15), "obj4 on cycle %d", text variable: GVL.obj[4], invisible if: GVL.obj[4]=0
    Rectangle (696,458 96x18), "trowing out", colour toggle: GVL.trowingObjectOut, invisible if: GVL.trowingObjectOut <> True
    Ellipse (483,214 30x30), colour toggle: GVL.topRight_IB
    Ellipse (289,214 30x30), colour toggle: GVL.topLeft_IB
    Ellipse (441,419 30x30), colour toggle: GVL.bottomRight_IB
    Ellipse (284,419 30x30), colour toggle: GVL.bottomLeft_IB
    Polygon (373,229) (412,204) (412,229) (412,239) (412,254), colour toggle: GVL.topBeltLeft_OB
        OnMouseDown: toggle GVL.topBeltLeft_OB
    Polygon (702,229) (741,204) (741,229) (741,239) (741,254), colour toggle: GVL.rightLiftBeltLeft_OB, invisible if: rightLiftUpPosition_IB <> True
        OnMouseDown: toggle GVL.rightLiftBeltLeft_OB
    Polygon (406,434) (367,409) (367,434) (367,444) (367,459), colour toggle: GVL.bottomBeltRight_OB
        OnMouseDown: toggle GVL.bottomBeltRight_OB
    Polygon (156,378) (128,339) (156,339) (168,339) (183,339), colour toggle: GVL.leftLiftDown_OB
        OnMouseDown: toggle GVL.leftLiftDown_OB
    Polygon (634,388) (606,349) (634,349) (646,349) (661,349), colour toggle: GVL.rightLiftDown_OB
        OnMouseDown: toggle GVL.rightLiftDown_OB
    Polygon (634,260) (606,299) (634,299) (646,299) (661,299), colour toggle: GVL.rightLiftUp_OB
        OnMouseDown: toggle GVL.rightLiftUp_OB
    Polygon (155,255) (127,294) (155,294) (167,294) (182,294), colour toggle: GVL.leftLiftUp_OB
        OnMouseDown: toggle GVL.leftLiftUp_OB
    Button (310,121 150x30), "Reset"
        OnMouseDown: toggle resetAll
        OnMouseUp: toggle resetAll
    Rectangle (208,159 469x24), "%s", text variable: errMessage, colour toggle: ERR <> 0, invisible if: ERR = 0
    Button (680,153 81x30), "Clear", invisible if: ERR = 0
        OnMouseDown: toggle resetError
    Rectangle (311,304 188x41), "%s", text variable: textMA, colour toggle: auto
        OnMouseDown: toggle auto
    Rectangle (632,247 15x15), "%d", text variable: GVL.topRightLiftExpArr[1], invisible if: GVL.topRightLiftExpArr[1] =0
    Rectangle (652,247 15x15), "%d", text variable: GVL.topRightLiftExpArr[2], invisible if: GVL.topRightLiftExpArr[2]=0
    Rectangle (672,247 15x15), "%d", text variable: GVL.topRightLiftExpArr[3], invisible if: GVL.topRightLiftExpArr[3] = 0
    Rectangle (692,247 15x15), "%d", text variable: GVL.topRightLiftExpArr[4], invisible if: GVL.topRightLiftExpArr[4]=0
    Rectangle (712,247 15x15), "%d", text variable: GVL.topRightLiftExpArr[5], invisible if: GVL.topRightLiftExpArr[5]=0
    Rectangle (506,198 15x15), "%d", text variable: GVL.topRightExpArr[1], invisible if: GVL.topRightExpArr[1]=0
    Rectangle (526,198 15x15), "%d", text variable: GVL.topRightExpArr[2], invisible if: GVL.topRightExpArr[2]=0
    Rectangle (546,198 15x15), "%d", text variable: GVL.topRightExpArr[3], invisible if: GVL.topRightExpArr[3]=0
    Rectangle (567,198 14x15), "%d", text variable: GVL.topRightExpArr[4], invisible if: GVL.topRightExpArr[4]=0
    Rectangle (588,199 15x15), "%d", text variable: GVL.topRightExpArr[5], invisible if: GVL.topRightExpArr[5]=0
    Rectangle (311,198 14x15), "%d", text variable: GVL.topLeftExpArr[1], invisible if: GVL.topLeftExpArr[1] = 0
    Rectangle (331,198 15x15), "%d", text variable: GVL.topLeftExpArr[2], invisible if: GVL.topLeftExpArr[2]=0
    Rectangle (351,198 15x15), "%d", text variable: GVL.topLeftExpArr[3], invisible if: GVL.topLeftExpArr[3]=0
    Rectangle (371,198 14x15), "%d", text variable: GVL.topLeftExpArr[4], invisible if: GVL.topLeftExpArr[4]=0
    Rectangle (391,198 15x15), "%d", text variable: GVL.topLeftExpArr[5], invisible if: GVL.topLeftExpArr[5]=0
    Rectangle (227,198 15x15), "%d", text variable: GVL.topLeftLiftExpArr[1], invisible if: GVL.topLeftLiftExpArr[1]=0
    Rectangle (247,198 15x15), "%d", text variable: GVL.topLeftLiftExpArr[2], invisible if: GVL.topLeftLiftExpArr[2]=0
    Rectangle (267,198 11x15), "%d", text variable: GVL.topLeftLiftExpArr[3], invisible if: GVL.topLeftLiftExpArr[3]=0
    Rectangle (287,198 14x15), "%d", text variable: GVL.topLeftLiftExpArr[4], invisible if: GVL.topLeftLiftExpArr[4]=0
    Rectangle (307,198 15x15), "%d", text variable: GVL.topLeftLiftExpArr[5], invisible if: GVL.topLeftLiftExpArr[5]=0
    Rectangle (65,397 15x15), "%d", text variable: GVL.bottomLeftLiftExpArr[1], invisible if: GVL.bottomLeftLiftExpArr[1]=0
    Rectangle (85,397 15x15), "%d", text variable: GVL.bottomLeftLiftExpArr[2], invisible if: GVL.bottomLeftLiftExpArr[2]=0
    Rectangle (105,397 15x15), "%d", text variable: GVL.bottomLeftLiftExpArr[3], invisible if: GVL.bottomLeftLiftExpArr[3]=0
    Rectangle (125,397 15x15), "%d", text variable: GVL.bottomLeftLiftExpArr[4], invisible if: GVL.bottomLeftLiftExpArr[4] = 0
    Rectangle (145,397 15x15), "%d", text variable: GVL.bottomLeftLiftExpArr[5], invisible if: GVL.bottomLeftLiftExpArr[5]=0
    Label (316,5 60x30), "Objects:"
    Ellipse (620,214 30x30), colour toggle: GVL.rightLiftOptical_IB, invisible if: rightLiftUpPosition_IB <> True
    Polygon (786,229) (747,204) (747,229) (747,239) (747,254), colour toggle: GVL.rightLiftBeltRight_OB, invisible if: rightLiftUpPosition_IB <> True
        OnMouseDown: toggle GVL.rightLiftBeltRight_OB
    RoundedRectangle (572,313 125x20), invisible if: rightLiftUpPosition_IB or rightLiftDownPosition_IB
    Polygon (702,323) (741,298) (741,323) (741,333) (741,348), colour toggle: GVL.rightLiftBeltLeft_OB, invisible if: rightLiftUpPosition_IB or rightLiftDownPosition_IB
        OnMouseDown: toggle GVL.rightLiftBeltLeft_OB
    Ellipse (620,308 30x30), colour toggle: GVL.rightLiftOptical_IB, invisible if: rightLiftUpPosition_IB or rightLiftDownPosition_IB
    Polygon (786,323) (747,298) (747,323) (747,333) (747,348), colour toggle: GVL.rightLiftBeltRight_OB, invisible if: rightLiftUpPosition_IB or rightLiftDownPosition_IB
        OnMouseDown: toggle GVL.rightLiftBeltRight_OB
    RoundedRectangle (576,423 125x20), invisible if: not rightLiftDownPosition_IB
    Polygon (706,433) (745,408) (745,433) (745,443) (745,458), colour toggle: GVL.rightLiftBeltLeft_OB, invisible if: not rightLiftDownPosition_IB
        OnMouseDown: toggle GVL.rightLiftBeltLeft_OB
    Ellipse (624,418 30x30), colour toggle: GVL.rightLiftOptical_IB, invisible if: not rightLiftDownPosition_IB
    Polygon (790,433) (751,408) (751,433) (751,443) (751,458), colour toggle: GVL.rightLiftBeltRight_OB, invisible if: not rightLiftDownPosition_IB
        OnMouseDown: toggle GVL.rightLiftBeltRight_OB
    RoundedRectangle (95,216 125x20), invisible if: not leftLiftUpPosition_IB
    Polygon (5,225) (44,200) (44,225) (44,235) (44,250), colour toggle: GVL.leftLiftBeltLeft_OB, invisible if: leftLiftUpPosition_IB <> True
        OnMouseDown: toggle GVL.leftLiftBeltLeft_OB
    Ellipse (143,211 30x30), colour toggle: GVL.leftLiftOptical_IB, invisible if: not leftLiftUpPosition_IB
    Polygon (89,225) (50,200) (50,225) (50,235) (50,250), colour toggle: GVL.leftLiftBeltRight_OB, invisible if: not leftLiftUpPosition_IB
        OnMouseDown: toggle GVL.leftLiftBeltRight_OB
    RoundedRectangle (95,307 125x20), invisible if: leftLiftUpPosition_IB or leftLiftDownPosition_IB
    Polygon (5,316) (44,291) (44,316) (44,326) (44,341), colour toggle: GVL.leftLiftBeltLeft_OB, invisible if: leftLiftUpPosition_IB or leftLiftDownPosition_IB
        OnMouseDown: toggle GVL.leftLiftBeltLeft_OB
    Ellipse (143,302 30x30), colour toggle: GVL.leftLiftOptical_IB, invisible if: leftLiftUpPosition_IB or leftLiftDownPosition_IB
    Polygon (89,316) (50,291) (50,316) (50,326) (50,341), colour toggle: GVL.leftLiftBeltRight_OB, invisible if: leftLiftUpPosition_IB or leftLiftDownPosition_IB
        OnMouseDown: toggle GVL.leftLiftBeltRight_OB
    RoundedRectangle (91,422 125x20), invisible if: not leftLiftDownPosition_IB
    Polygon (1,431) (40,406) (40,431) (40,441) (40,456), colour toggle: GVL.leftLiftBeltLeft_OB, invisible if: not leftLiftDownPosition_IB
        OnMouseDown: toggle GVL.leftLiftBeltLeft_OB
    Ellipse (139,417 30x30), colour toggle: GVL.leftLiftOptical_IB, invisible if: not leftLiftDownPosition_IB
    Polygon (85,431) (46,406) (46,431) (46,441) (46,456), colour toggle: GVL.leftLiftBeltRight_OB, invisible if: not leftLiftDownPosition_IB
        OnMouseDown: toggle GVL.leftLiftBeltRight_OB
    Rectangle (194,398 15x15), "%d", text variable: GVL.bottomLeftExpArr[5], invisible if: GVL.bottomLeftExpArr[5]=0
    Rectangle (214,398 15x15), "%d", text variable: GVL.bottomLeftExpArr[4], invisible if: GVL.bottomLeftExpArr[4]=0
    Rectangle (234,398 15x15), "%d", text variable: GVL.bottomLeftExpArr[3], invisible if: GVL.bottomLeftExpArr[3]=0
    Rectangle (254,398 15x15), "%d", text variable: GVL.bottomLeftExpArr[2], invisible if: GVL.bottomLeftExpArr[2]=0
    Rectangle (274,398 15x15), "%d", text variable: GVL.bottomLeftExpArr[1], invisible if: GVL.bottomLeftExpArr[1]=0
    Rectangle (351,401 15x15), "%d", text variable: GVL.bottomRightExpArr[5], invisible if: GVL.bottomRightExpArr[5]=0
    Rectangle (371,401 15x15), "%d", text variable: GVL.bottomRightExpArr[4], invisible if: GVL.bottomRightExpArr[4]=0
    Rectangle (391,401 15x15), "%d", text variable: GVL.bottomRightExpArr[3], invisible if: GVL.bottomRightExpArr[3]=0
    Rectangle (411,401 15x15), "%d", text variable: GVL.bottomRightExpArr[2], invisible if: GVL.bottomRightExpArr[2]=0
    Rectangle (431,401 15x15), "%d", text variable: GVL.bottomRightExpArr[1], invisible if: GVL.bottomRightExpArr[1]=0
    Rectangle (470,405 15x15), "%d", text variable: GVL.bottomRightLiftExpArr[5], invisible if: GVL.bottomRightLiftExpArr[5]=0
    Rectangle (490,405 15x15), "%d", text variable: GVL.bottomRightLiftExpArr[4], invisible if: GVL.bottomRightLiftExpArr[4]=0
    Rectangle (510,405 15x15), "%d", text variable: GVL.bottomRightLiftExpArr[3], invisible if: GVL.bottomRightLiftExpArr[3]=0
    Rectangle (530,405 15x15), "%d", text variable: GVL.bottomRightLiftExpArr[2], invisible if: GVL.bottomRightLiftExpArr[2]=0
    Rectangle (550,405 15x15), "%d", text variable: GVL.bottomRightLiftExpArr[1], invisible if: GVL.bottomRightLiftExpArr[1]=0
END_VISUALIZATION
